TYPE InertiaEmulation_Struct :
UNION
		Value : INT;
		Bits : Bits_InertiaEmulation;
END_UNION
END_TYPE

(* stored: Version 1.1.0.1, ProductVersion 3.1.4022.18
   DUT InertiaEmulation_Struct: Id {29a4f158-423e-4985-b376-22da71d3fa49} *)
